FUNCTION_BLOCK FB_Conveyor
VAR_INPUT
	bManualMode:BOOL;
	bMoveRequest:BOOL;
	bEN_FeedbackError: BOOL;
END_VAR
VAR_OUTPUT
END_VAR
VAR
	bI_ConveyorOnFeedback AT %I*: BOOL;
	iQ_ConveyorSpeedOut	AT %Q*: INT;
	fbFeedbackErrorTON: TON;
	bOnCmd : BOOL;
	bManualOnCmd:BOOL;

	fbAnalogScale: fbAnalogMeasurement;
	stMeasureScaling: stMeasurementScalingData;
	fbMoveRequest_RTRIG: R_TRIG;
	fbCmdOnTOF: TOF;
END_VAR
VAR PERSISTENT
	rSpeedSet: REAL;
END_VAR

fbFeedbackErrorTON(IN:= (prIsON XOR bOnCmd) AND bEN_FeedbackError, PT:= T#10S);
stMeasureScaling.rScalingRawValue_II:=100.0;
stMeasureScaling.rScalingEngValue_I:=3000;
stMeasureScaling.rScalingEngValue_II:=32767;
fbAnalogScale(rIn:=rSpeedSet, stMeasureScalingData:=stMeasureScaling, tStalaCzasowa:=T#10MS);

bManualOnCmd R= NOT bManualMode;

fbMoveRequest_RTRIG(CLK:=bMoveRequest);
fbCmdOnTOF(IN:=fbMoveRequest_RTRIG.Q,PT:=T#10M);



IF bManualMode THEN
	prIsOn := bManualOnCmd;
ELSE
	prIsOn := fbCmdOnTOF.Q;
END_IF
IF bOnCmd THEN
	rSpeedSet := MAX(10,rSpeedSet);
	iQ_ConveyorSpeedOut := REAL_TO_INT(fbAnalogScale.rOutFiltered);
ELSE
	iQ_ConveyorSpeedOut := 3000;
END_IF

bMoveRequest:=FALSE;

PROPERTY prError : BOOL
GET
prError := fbFeedbackErrorTON.Q;
END_GET
END_PROPERTY

PROPERTY prIsOn : BOOL
GET
prIsOn := bI_ConveyorOnFeedback;
END_GET
SET
bOnCmd:=prIsOn;
END_SET
END_PROPERTY

PROPERTY prManualOn : BOOL
GET
END_GET
SET
END_SET
END_PROPERTY

END_FUNCTION_BLOCK

(* stored: Version 1.1.0.1, ProductVersion 3.1.4024.15
   POU FB_Conveyor: Id {0a89ffbc-5ceb-4c01-b8f9-acffc29e7ab7}, SpecialFunc None
   Property prError: Id {6211ab18-3897-447f-8a22-686b0fc90b82}
   Get Get: Id {041030bb-5e4f-4475-97a0-29ce58425d9e}
   Property prIsOn: Id {2cd67af5-4b4f-4081-921a-ffe719d45cf6}
   Get Get: Id {11d81eff-1fff-4c07-8023-235abb4321ed}
   Set Set: Id {198b1ee6-e006-48a3-8d6e-85aec495f8ce}
   Property prManualOn: Id {6a98c453-4184-41b7-aa63-942367f27205}
   Get Get: Id {274179ae-fc59-4459-a3cb-33732cc845e0}
   Set Set: Id {37a3c3ec-3fa8-4b08-b891-cb67d786e1f3} *)
